TYPE BIT8_ARRAY :
STRUCT
	bit0 : BIT;
	bit1 : BIT;
	bit2 : BIT;
	bit3 : BIT;
	bit4 : BIT;
	bit5 : BIT;
	bit6 : BIT;
	bit7 : BIT;
END_STRUCT
END_TYPE

(* stored: Version 1.1.0.1, ProductVersion 3.1.4024.11
   DUT BIT8_ARRAY: Id {20687552-5645-4eeb-8532-e3a7ded8b42e} *)
